// TIA Portal V17 export
// export: Created 2025-03-10T13:12:49.470688Z, ExportSetting WithDefaults, DisplayName Totally Integrated Automation Portal, DisplayVersion V17 Update 8, DisplayName TIA Portal Openness, DisplayVersion V17 Update 8, DisplayName TIA Portal Version Control Interface, DisplayVersion V17, DisplayName SINAMICS Startdrive Advanced, DisplayVersion V17 SP2, DisplayName SINAMICS Startdrive G110M, G120, G120C, G120D, G120P, G115D, DisplayVersion V17 SP2, DisplayName SINAMICS Startdrive G130, G150, S120, S150, SINAMICS MV, S210, DisplayVersion V17 SP2, DisplayName STEP 7 Professional, DisplayVersion V17 Update 8, DisplayName SINUMERIK ONE STEP 7 Toolbox, DisplayVersion V17 Update 12, DisplayName SINUMERIK 840D sl STEP 7 Toolbox, DisplayVersion V17 Update 12, DisplayName STEP 7 Safety, DisplayVersion V17 Update 6, DisplayName WinCC Advanced, DisplayVersion V17 Update 8
FUNCTION_BLOCK "FB21012_POWDER_FEEDER_HEATER_JKT"   // FB21012, LAD
TITLE = FB21012 POWDER FEEDER HEATER JKT
{ S7_Optimized_Access := 'FALSE' }
VERSION : 0.1
// stored: AutoNumber false, IsIECCheckEnabled false, SetENOAutomatically false, UDAEnableTagReadback false
   VAR_INPUT
      iPF_HEAT_AVAILABLE_OPTION : Bool;
      iPF_PROFINET_MODE_ACTIVE_FAULT : Bool;
      iPF_HOPPER_TEMP_GrHH_LINE_1 : Bool;   // POWDER FEEDER HOPPER TEMPERATURE LINE 1 ALARM
      iPF_HOPPER_TEMP_GrHH_LINE_2 : Bool;   // POWDER FEEDER HOPPER TEMPERATURE LINE 2 ALARM
      iCONTROL_ON_DELAYED : Bool;   // LOCAL MACHINE ON
      iAUTO_START_REQUEST : Bool;   // AUTO START REQUEST
      iAUTO_STOP_REQUEST : Bool;   // AUTO STOP SEQUEST
      iUNIT_NUMBER : Byte;
      iMANUAL_START_REQ_LINE_1 : Bool;
      iMANUAL_START_REQ_LINE_2 : Bool;
      iMANUAL_STOP_REQ_LINE_1 : Bool;
      iMANUAL_STOP_REQ_LINE_2 : Bool;
   END_VAR
   VAR_OUTPUT
      oPF_HEATING_ON_CMD_LINE_1 : Bool;   // POWDER FEEDER HEATING ON COMMAND LINE 1
      oPF_HEATING_ON_CMD_LINE_2 : Bool;   // POWDER FEEDER HEATING ON COMMAND LINE 2
      oPF_HEATING_OFF_CMD_LINE_1 : Bool;   // POWDER FEEDER HEATING OF COMMAND LINE 1
      oPF_HEATING_OFF_CMD_LINE_2 : Bool;   // POWDER FEEDER HEATING OF COMMAND LINE 2
      oSWITCHONCONDITION_ON_LINE_1 : Bool;
      oSWITCHONCONDITION_ON_LINE_2 : Bool;
      oSWITCHONCONDITION_OFF_LINE_1 : Bool;
      oSWITCHONCONDITION_OFF_LINE_2 : Bool;
      oMOTION_ACTIVE_RIGHT_LINE_1 : Bool;
      oMOTION_ACTIVE_RIGHT_LINE_2 : Bool;
      oMOTION_ACTIVE_LEFT_LINE_1 : Bool;
      oMOTION_ACTIVE_LEFT_LINE_2 : Bool;
      oLIMIT_RIGHT_LINE_1 : Bool;
      oLIMIT_RIGHT_LINE_2 : Bool;
      oLIMIT_LEFT_LINE_1 : Bool;
      oLIMIT_LEFT_LINE_2 : Bool;
      oALARM_HOPPER_LINE_1_TEMP_ABOVE_HIGH_LIMIT : Bool;
      oALARM_HOPPER_LINE_2_TEMP_ABOVE_HIGH_LIMIT : Bool;
   END_VAR
   VAR DB_SPECIFIC
      DATA : "POWDER FEEDER HEATER JKT";
      INPUT_SETTINGS : Struct
         UNIT_NUMBER : Int;
         FEEDER_NUMBER : Int;
      END_STRUCT;
      HEATER_STATUS_LINE_1 { S7_SetPoint := 'True'} : Byte;
      HEATER_STATUS_LINE_2 : Byte;
   END_VAR
   VAR_TEMP
      DB_NUMBER : DInt;
   END_VAR
   VAR_TEMP   // added for the SCL form of the ladder/FBD networks
      _w1 : Bool;
      _w2 : Bool;
   END_VAR
BEGIN

NETWORK
TITLE = READ INSTANCE DB NUMBER
      L     DINO;
      +     10#800000;
      T     #DB_NUMBER;

REGION Network 2: START GENERAL CONDITIONS / Start General Conditions
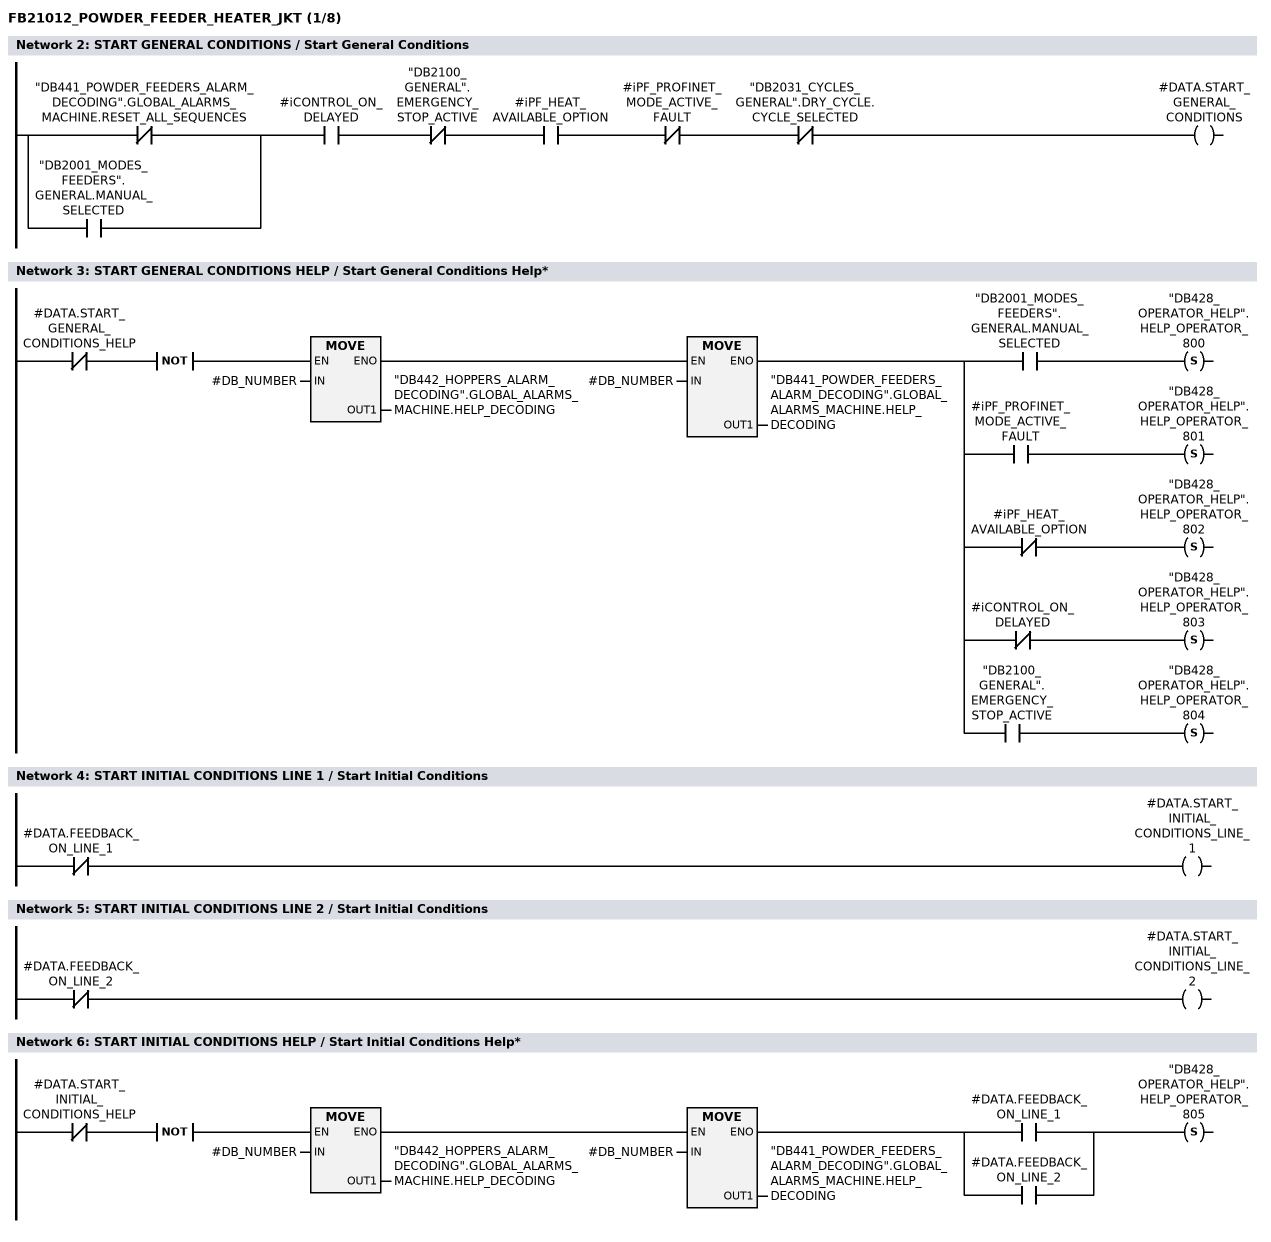
   RUNG wire#powerrail
      I_Contact( "DB441_POWDER_FEEDERS_ALARM_DECODING".GLOBAL_ALARMS_MACHINE.RESET_ALL_SEQUENCES )
      wire#w1
      Contact( #iCONTROL_ON_DELAYED )
      I_Contact( "DB2100_GENERAL".EMERGENCY_STOP_ACTIVE )
      Contact( #iPF_HEAT_AVAILABLE_OPTION )
      I_Contact( #iPF_PROFINET_MODE_ACTIVE_FAULT )
      I_Contact( "DB2031_CYCLES_GENERAL".DRY_CYCLE.CYCLE_SELECTED )
      Coil( #DATA.START_GENERAL_CONDITIONS )
   END_RUNG
   RUNG wire#powerrail
      Contact( "DB2001_MODES_FEEDERS".GENERAL.MANUAL_SELECTED )
   END_RUNG wire#w1
   // the same network as SCL:
   #DATA.START_GENERAL_CONDITIONS := (NOT "DB441_POWDER_FEEDERS_ALARM_DECODING".GLOBAL_ALARMS_MACHINE.RESET_ALL_SEQUENCES OR "DB2001_MODES_FEEDERS".GENERAL.MANUAL_SELECTED) AND #iCONTROL_ON_DELAYED AND NOT "DB2100_GENERAL".EMERGENCY_STOP_ACTIVE AND #iPF_HEAT_AVAILABLE_OPTION AND NOT #iPF_PROFINET_MODE_ACTIVE_FAULT AND NOT "DB2031_CYCLES_GENERAL".DRY_CYCLE.CYCLE_SELECTED;
END_REGION

REGION Network 3: START GENERAL CONDITIONS HELP / Start General Conditions Help*
   RUNG wire#powerrail
      I_Contact( #DATA.START_GENERAL_CONDITIONS_HELP )
      Not()
      Move(in := #DB_NUMBER, out1 => "DB442_HOPPERS_ALARM_DECODING".GLOBAL_ALARMS_MACHINE.HELP_DECODING)
      Move(in := #DB_NUMBER, out1 => "DB441_POWDER_FEEDERS_ALARM_DECODING".GLOBAL_ALARMS_MACHINE.HELP_DECODING)
      wire#w1
      Contact( "DB2001_MODES_FEEDERS".GENERAL.MANUAL_SELECTED )
      S_Coil( "DB428_OPERATOR_HELP".HELP_OPERATOR_800 )
   END_RUNG
   RUNG wire#w1
      Contact( #iPF_PROFINET_MODE_ACTIVE_FAULT )
      S_Coil( "DB428_OPERATOR_HELP".HELP_OPERATOR_801 )
   END_RUNG
   RUNG wire#w1
      I_Contact( #iPF_HEAT_AVAILABLE_OPTION )
      S_Coil( "DB428_OPERATOR_HELP".HELP_OPERATOR_802 )
   END_RUNG
   RUNG wire#w1
      I_Contact( #iCONTROL_ON_DELAYED )
      S_Coil( "DB428_OPERATOR_HELP".HELP_OPERATOR_803 )
   END_RUNG
   RUNG wire#w1
      Contact( "DB2100_GENERAL".EMERGENCY_STOP_ACTIVE )
      S_Coil( "DB428_OPERATOR_HELP".HELP_OPERATOR_804 )
   END_RUNG
   // the same network as SCL:
   #_w1 := NOT (NOT #DATA.START_GENERAL_CONDITIONS_HELP);
   IF #_w1 THEN
       "DB442_HOPPERS_ALARM_DECODING".GLOBAL_ALARMS_MACHINE.HELP_DECODING := #DB_NUMBER;
       "DB441_POWDER_FEEDERS_ALARM_DECODING".GLOBAL_ALARMS_MACHINE.HELP_DECODING := #DB_NUMBER;
   END_IF;
   IF #_w1 AND "DB2001_MODES_FEEDERS".GENERAL.MANUAL_SELECTED THEN
       "DB428_OPERATOR_HELP".HELP_OPERATOR_800 := TRUE;
   END_IF;
   IF #_w1 AND #iPF_PROFINET_MODE_ACTIVE_FAULT THEN "DB428_OPERATOR_HELP".HELP_OPERATOR_801 := TRUE; END_IF;
   IF #_w1 AND NOT #iPF_HEAT_AVAILABLE_OPTION THEN "DB428_OPERATOR_HELP".HELP_OPERATOR_802 := TRUE; END_IF;
   IF #_w1 AND NOT #iCONTROL_ON_DELAYED THEN "DB428_OPERATOR_HELP".HELP_OPERATOR_803 := TRUE; END_IF;
   IF #_w1 AND "DB2100_GENERAL".EMERGENCY_STOP_ACTIVE THEN
       "DB428_OPERATOR_HELP".HELP_OPERATOR_804 := TRUE;
   END_IF;
END_REGION

REGION Network 4: START INITIAL CONDITIONS LINE 1 / Start Initial Conditions
   RUNG wire#powerrail
      I_Contact( #DATA.FEEDBACK_ON_LINE_1 )
      Coil( #DATA.START_INITIAL_CONDITIONS_LINE_1 )
   END_RUNG
   // the same network as SCL:
   #DATA.START_INITIAL_CONDITIONS_LINE_1 := NOT #DATA.FEEDBACK_ON_LINE_1;
END_REGION

REGION Network 5: START INITIAL CONDITIONS LINE 2 / Start Initial Conditions
   RUNG wire#powerrail
      I_Contact( #DATA.FEEDBACK_ON_LINE_2 )
      Coil( #DATA.START_INITIAL_CONDITIONS_LINE_2 )
   END_RUNG
   // the same network as SCL:
   #DATA.START_INITIAL_CONDITIONS_LINE_2 := NOT #DATA.FEEDBACK_ON_LINE_2;
END_REGION

REGION Network 6: START INITIAL CONDITIONS HELP / Start Initial Conditions Help*
   RUNG wire#powerrail
      I_Contact( #DATA.START_INITIAL_CONDITIONS_HELP )
      Not()
      Move(in := #DB_NUMBER, out1 => "DB442_HOPPERS_ALARM_DECODING".GLOBAL_ALARMS_MACHINE.HELP_DECODING)
      Move(in := #DB_NUMBER, out1 => "DB441_POWDER_FEEDERS_ALARM_DECODING".GLOBAL_ALARMS_MACHINE.HELP_DECODING)
      wire#w1
      Contact( #DATA.FEEDBACK_ON_LINE_1 )
      wire#w2
      S_Coil( "DB428_OPERATOR_HELP".HELP_OPERATOR_805 )
   END_RUNG
   RUNG wire#w1
      Contact( #DATA.FEEDBACK_ON_LINE_2 )
   END_RUNG wire#w2
   // the same network as SCL:
   #_w1 := NOT (NOT #DATA.START_INITIAL_CONDITIONS_HELP);
   IF #_w1 THEN
       "DB442_HOPPERS_ALARM_DECODING".GLOBAL_ALARMS_MACHINE.HELP_DECODING := #DB_NUMBER;
       "DB441_POWDER_FEEDERS_ALARM_DECODING".GLOBAL_ALARMS_MACHINE.HELP_DECODING := #DB_NUMBER;
   END_IF;
   IF #_w1 AND (#DATA.FEEDBACK_ON_LINE_1 OR #DATA.FEEDBACK_ON_LINE_2) THEN
       "DB428_OPERATOR_HELP".HELP_OPERATOR_805 := TRUE;
   END_IF;
END_REGION

REGION Network 7: MANUAL MODE NOT SELECTED HELP / Manual Mode Not Selected Help*
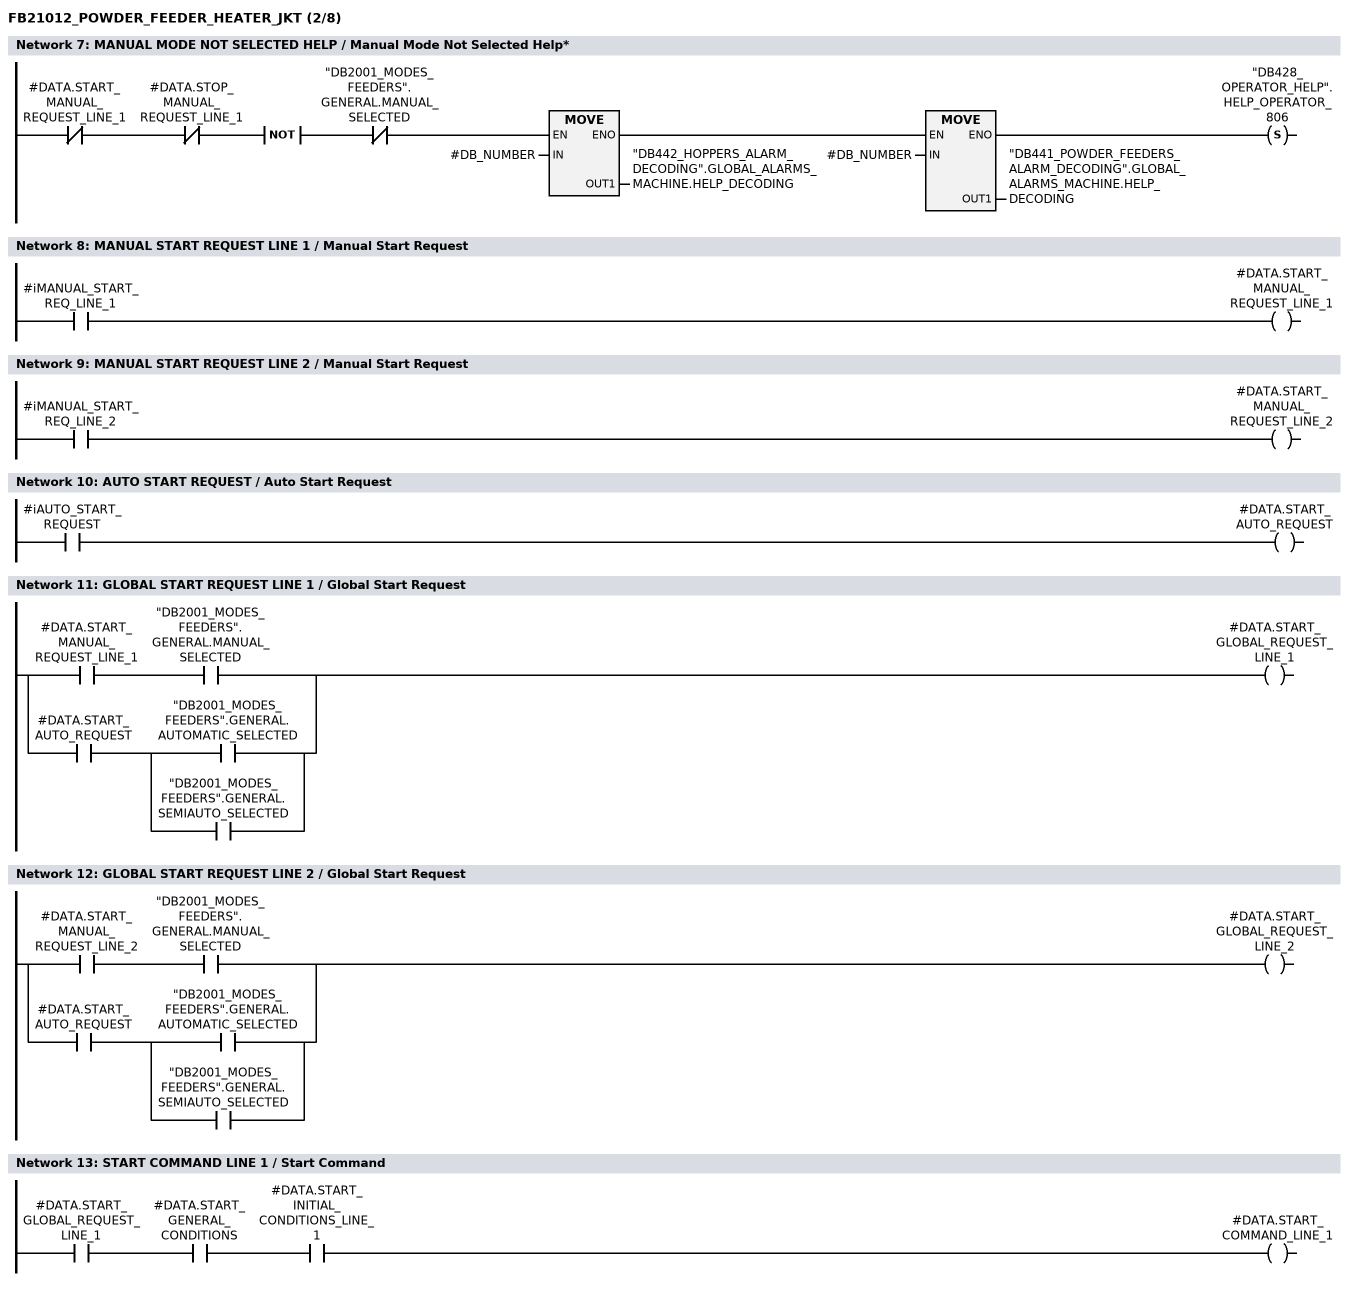
   RUNG wire#powerrail
      I_Contact( #DATA.START_MANUAL_REQUEST_LINE_1 )
      I_Contact( #DATA.STOP_MANUAL_REQUEST_LINE_1 )
      Not()
      I_Contact( "DB2001_MODES_FEEDERS".GENERAL.MANUAL_SELECTED )
      Move(in := #DB_NUMBER, out1 => "DB442_HOPPERS_ALARM_DECODING".GLOBAL_ALARMS_MACHINE.HELP_DECODING)
      Move(in := #DB_NUMBER, out1 => "DB441_POWDER_FEEDERS_ALARM_DECODING".GLOBAL_ALARMS_MACHINE.HELP_DECODING)
      S_Coil( "DB428_OPERATOR_HELP".HELP_OPERATOR_806 )
   END_RUNG
   // the same network as SCL:
   IF NOT (NOT #DATA.START_MANUAL_REQUEST_LINE_1 AND NOT #DATA.STOP_MANUAL_REQUEST_LINE_1) AND NOT "DB2001_MODES_FEEDERS".GENERAL.MANUAL_SELECTED THEN
       "DB442_HOPPERS_ALARM_DECODING".GLOBAL_ALARMS_MACHINE.HELP_DECODING := #DB_NUMBER;
       "DB441_POWDER_FEEDERS_ALARM_DECODING".GLOBAL_ALARMS_MACHINE.HELP_DECODING := #DB_NUMBER;
       "DB428_OPERATOR_HELP".HELP_OPERATOR_806 := TRUE;
   END_IF;
END_REGION

REGION Network 8: MANUAL START REQUEST LINE 1 / Manual Start Request
   RUNG wire#powerrail
      Contact( #iMANUAL_START_REQ_LINE_1 )
      Coil( #DATA.START_MANUAL_REQUEST_LINE_1 )
   END_RUNG
   // the same network as SCL:
   #DATA.START_MANUAL_REQUEST_LINE_1 := #iMANUAL_START_REQ_LINE_1;
END_REGION

REGION Network 9: MANUAL START REQUEST LINE 2 / Manual Start Request
   RUNG wire#powerrail
      Contact( #iMANUAL_START_REQ_LINE_2 )
      Coil( #DATA.START_MANUAL_REQUEST_LINE_2 )
   END_RUNG
   // the same network as SCL:
   #DATA.START_MANUAL_REQUEST_LINE_2 := #iMANUAL_START_REQ_LINE_2;
END_REGION

REGION Network 10: AUTO START REQUEST / Auto Start Request
   RUNG wire#powerrail
      Contact( #iAUTO_START_REQUEST )
      Coil( #DATA.START_AUTO_REQUEST )
   END_RUNG
   // the same network as SCL:
   #DATA.START_AUTO_REQUEST := #iAUTO_START_REQUEST;
END_REGION

REGION Network 11: GLOBAL START REQUEST LINE 1 / Global Start Request
   RUNG wire#powerrail
      Contact( #DATA.START_MANUAL_REQUEST_LINE_1 )
      Contact( "DB2001_MODES_FEEDERS".GENERAL.MANUAL_SELECTED )
      wire#w1
      Coil( #DATA.START_GLOBAL_REQUEST_LINE_1 )
   END_RUNG
   RUNG wire#powerrail
      Contact( #DATA.START_AUTO_REQUEST )
      wire#w2
      Contact( "DB2001_MODES_FEEDERS".GENERAL.AUTOMATIC_SELECTED )
   END_RUNG wire#w1
   RUNG wire#w2
      Contact( "DB2001_MODES_FEEDERS".GENERAL.SEMIAUTO_SELECTED )
   END_RUNG wire#w1
   // the same network as SCL:
   #DATA.START_GLOBAL_REQUEST_LINE_1 := (#DATA.START_MANUAL_REQUEST_LINE_1 AND "DB2001_MODES_FEEDERS".GENERAL.MANUAL_SELECTED) OR (#DATA.START_AUTO_REQUEST AND ("DB2001_MODES_FEEDERS".GENERAL.AUTOMATIC_SELECTED OR "DB2001_MODES_FEEDERS".GENERAL.SEMIAUTO_SELECTED));
END_REGION

REGION Network 12: GLOBAL START REQUEST LINE 2 / Global Start Request
   RUNG wire#powerrail
      Contact( #DATA.START_MANUAL_REQUEST_LINE_2 )
      Contact( "DB2001_MODES_FEEDERS".GENERAL.MANUAL_SELECTED )
      wire#w1
      Coil( #DATA.START_GLOBAL_REQUEST_LINE_2 )
   END_RUNG
   RUNG wire#powerrail
      Contact( #DATA.START_AUTO_REQUEST )
      wire#w2
      Contact( "DB2001_MODES_FEEDERS".GENERAL.AUTOMATIC_SELECTED )
   END_RUNG wire#w1
   RUNG wire#w2
      Contact( "DB2001_MODES_FEEDERS".GENERAL.SEMIAUTO_SELECTED )
   END_RUNG wire#w1
   // the same network as SCL:
   #DATA.START_GLOBAL_REQUEST_LINE_2 := (#DATA.START_MANUAL_REQUEST_LINE_2 AND "DB2001_MODES_FEEDERS".GENERAL.MANUAL_SELECTED) OR (#DATA.START_AUTO_REQUEST AND ("DB2001_MODES_FEEDERS".GENERAL.AUTOMATIC_SELECTED OR "DB2001_MODES_FEEDERS".GENERAL.SEMIAUTO_SELECTED));
END_REGION

REGION Network 13: START COMMAND LINE 1 / Start Command
   RUNG wire#powerrail
      Contact( #DATA.START_GLOBAL_REQUEST_LINE_1 )
      Contact( #DATA.START_GENERAL_CONDITIONS )
      Contact( #DATA.START_INITIAL_CONDITIONS_LINE_1 )
      Coil( #DATA.START_COMMAND_LINE_1 )
   END_RUNG
   // the same network as SCL:
   #DATA.START_COMMAND_LINE_1 := #DATA.START_GLOBAL_REQUEST_LINE_1 AND #DATA.START_GENERAL_CONDITIONS AND #DATA.START_INITIAL_CONDITIONS_LINE_1;
END_REGION

REGION Network 14: START COMMAND LINE 2 / Start Command
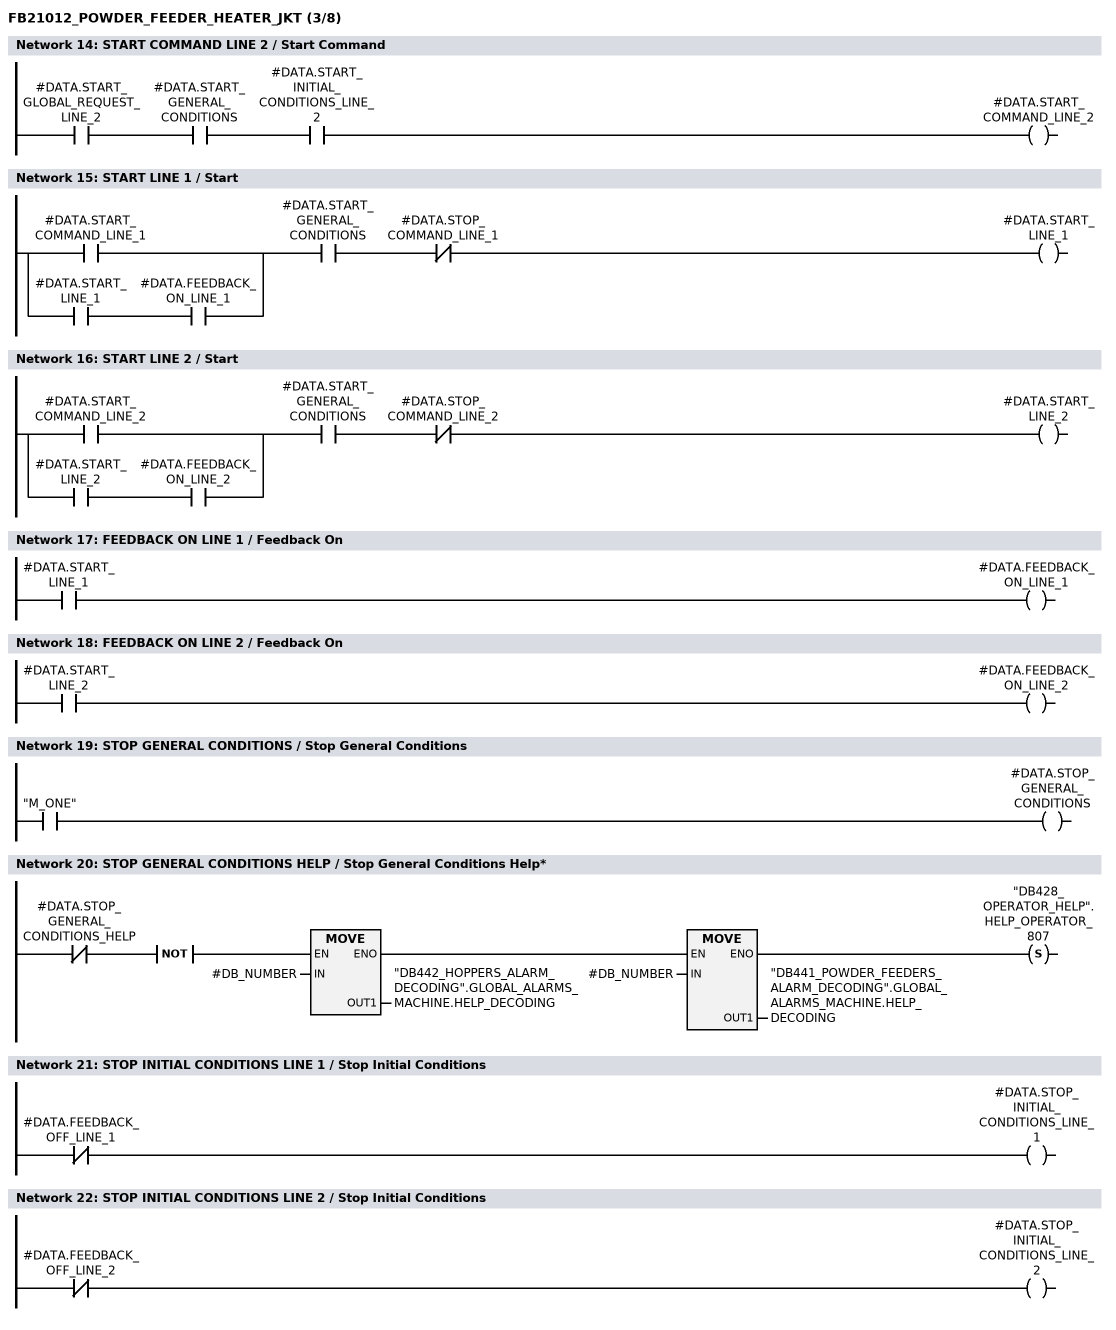
   RUNG wire#powerrail
      Contact( #DATA.START_GLOBAL_REQUEST_LINE_2 )
      Contact( #DATA.START_GENERAL_CONDITIONS )
      Contact( #DATA.START_INITIAL_CONDITIONS_LINE_2 )
      Coil( #DATA.START_COMMAND_LINE_2 )
   END_RUNG
   // the same network as SCL:
   #DATA.START_COMMAND_LINE_2 := #DATA.START_GLOBAL_REQUEST_LINE_2 AND #DATA.START_GENERAL_CONDITIONS AND #DATA.START_INITIAL_CONDITIONS_LINE_2;
END_REGION

REGION Network 15: START LINE 1 / Start
   RUNG wire#powerrail
      Contact( #DATA.START_COMMAND_LINE_1 )
      wire#w1
      Contact( #DATA.START_GENERAL_CONDITIONS )
      I_Contact( #DATA.STOP_COMMAND_LINE_1 )
      Coil( #DATA.START_LINE_1 )
   END_RUNG
   RUNG wire#powerrail
      Contact( #DATA.START_LINE_1 )
      Contact( #DATA.FEEDBACK_ON_LINE_1 )
   END_RUNG wire#w1
   // the same network as SCL:
   #DATA.START_LINE_1 := (#DATA.START_COMMAND_LINE_1 OR (#DATA.START_LINE_1 AND #DATA.FEEDBACK_ON_LINE_1)) AND #DATA.START_GENERAL_CONDITIONS AND NOT #DATA.STOP_COMMAND_LINE_1;
END_REGION

REGION Network 16: START LINE 2 / Start
   RUNG wire#powerrail
      Contact( #DATA.START_COMMAND_LINE_2 )
      wire#w1
      Contact( #DATA.START_GENERAL_CONDITIONS )
      I_Contact( #DATA.STOP_COMMAND_LINE_2 )
      Coil( #DATA.START_LINE_2 )
   END_RUNG
   RUNG wire#powerrail
      Contact( #DATA.START_LINE_2 )
      Contact( #DATA.FEEDBACK_ON_LINE_2 )
   END_RUNG wire#w1
   // the same network as SCL:
   #DATA.START_LINE_2 := (#DATA.START_COMMAND_LINE_2 OR (#DATA.START_LINE_2 AND #DATA.FEEDBACK_ON_LINE_2)) AND #DATA.START_GENERAL_CONDITIONS AND NOT #DATA.STOP_COMMAND_LINE_2;
END_REGION

REGION Network 17: FEEDBACK ON LINE 1 / Feedback On
   RUNG wire#powerrail
      Contact( #DATA.START_LINE_1 )
      Coil( #DATA.FEEDBACK_ON_LINE_1 )
   END_RUNG
   // the same network as SCL:
   #DATA.FEEDBACK_ON_LINE_1 := #DATA.START_LINE_1;
END_REGION

REGION Network 18: FEEDBACK ON LINE 2 / Feedback On
   RUNG wire#powerrail
      Contact( #DATA.START_LINE_2 )
      Coil( #DATA.FEEDBACK_ON_LINE_2 )
   END_RUNG
   // the same network as SCL:
   #DATA.FEEDBACK_ON_LINE_2 := #DATA.START_LINE_2;
END_REGION

REGION Network 19: STOP GENERAL CONDITIONS / Stop General Conditions
   RUNG wire#powerrail
      Contact( "M_ONE" )
      Coil( #DATA.STOP_GENERAL_CONDITIONS )
   END_RUNG
   // the same network as SCL:
   #DATA.STOP_GENERAL_CONDITIONS := "M_ONE";
END_REGION

REGION Network 20: STOP GENERAL CONDITIONS HELP / Stop General Conditions Help*
   RUNG wire#powerrail
      I_Contact( #DATA.STOP_GENERAL_CONDITIONS_HELP )
      Not()
      Move(in := #DB_NUMBER, out1 => "DB442_HOPPERS_ALARM_DECODING".GLOBAL_ALARMS_MACHINE.HELP_DECODING)
      Move(in := #DB_NUMBER, out1 => "DB441_POWDER_FEEDERS_ALARM_DECODING".GLOBAL_ALARMS_MACHINE.HELP_DECODING)
      S_Coil( "DB428_OPERATOR_HELP".HELP_OPERATOR_807 )
   END_RUNG
   // the same network as SCL:
   IF NOT (NOT #DATA.STOP_GENERAL_CONDITIONS_HELP) THEN
       "DB442_HOPPERS_ALARM_DECODING".GLOBAL_ALARMS_MACHINE.HELP_DECODING := #DB_NUMBER;
       "DB441_POWDER_FEEDERS_ALARM_DECODING".GLOBAL_ALARMS_MACHINE.HELP_DECODING := #DB_NUMBER;
       "DB428_OPERATOR_HELP".HELP_OPERATOR_807 := TRUE;
   END_IF;
END_REGION

REGION Network 21: STOP INITIAL CONDITIONS LINE 1 / Stop Initial Conditions
   RUNG wire#powerrail
      I_Contact( #DATA.FEEDBACK_OFF_LINE_1 )
      Coil( #DATA.STOP_INITIAL_CONDITIONS_LINE_1 )
   END_RUNG
   // the same network as SCL:
   #DATA.STOP_INITIAL_CONDITIONS_LINE_1 := NOT #DATA.FEEDBACK_OFF_LINE_1;
END_REGION

REGION Network 22: STOP INITIAL CONDITIONS LINE 2 / Stop Initial Conditions
   RUNG wire#powerrail
      I_Contact( #DATA.FEEDBACK_OFF_LINE_2 )
      Coil( #DATA.STOP_INITIAL_CONDITIONS_LINE_2 )
   END_RUNG
   // the same network as SCL:
   #DATA.STOP_INITIAL_CONDITIONS_LINE_2 := NOT #DATA.FEEDBACK_OFF_LINE_2;
END_REGION

REGION Network 23: STOP INITIAL CONDITIONS HELP / Stop Initial Conditions Help*
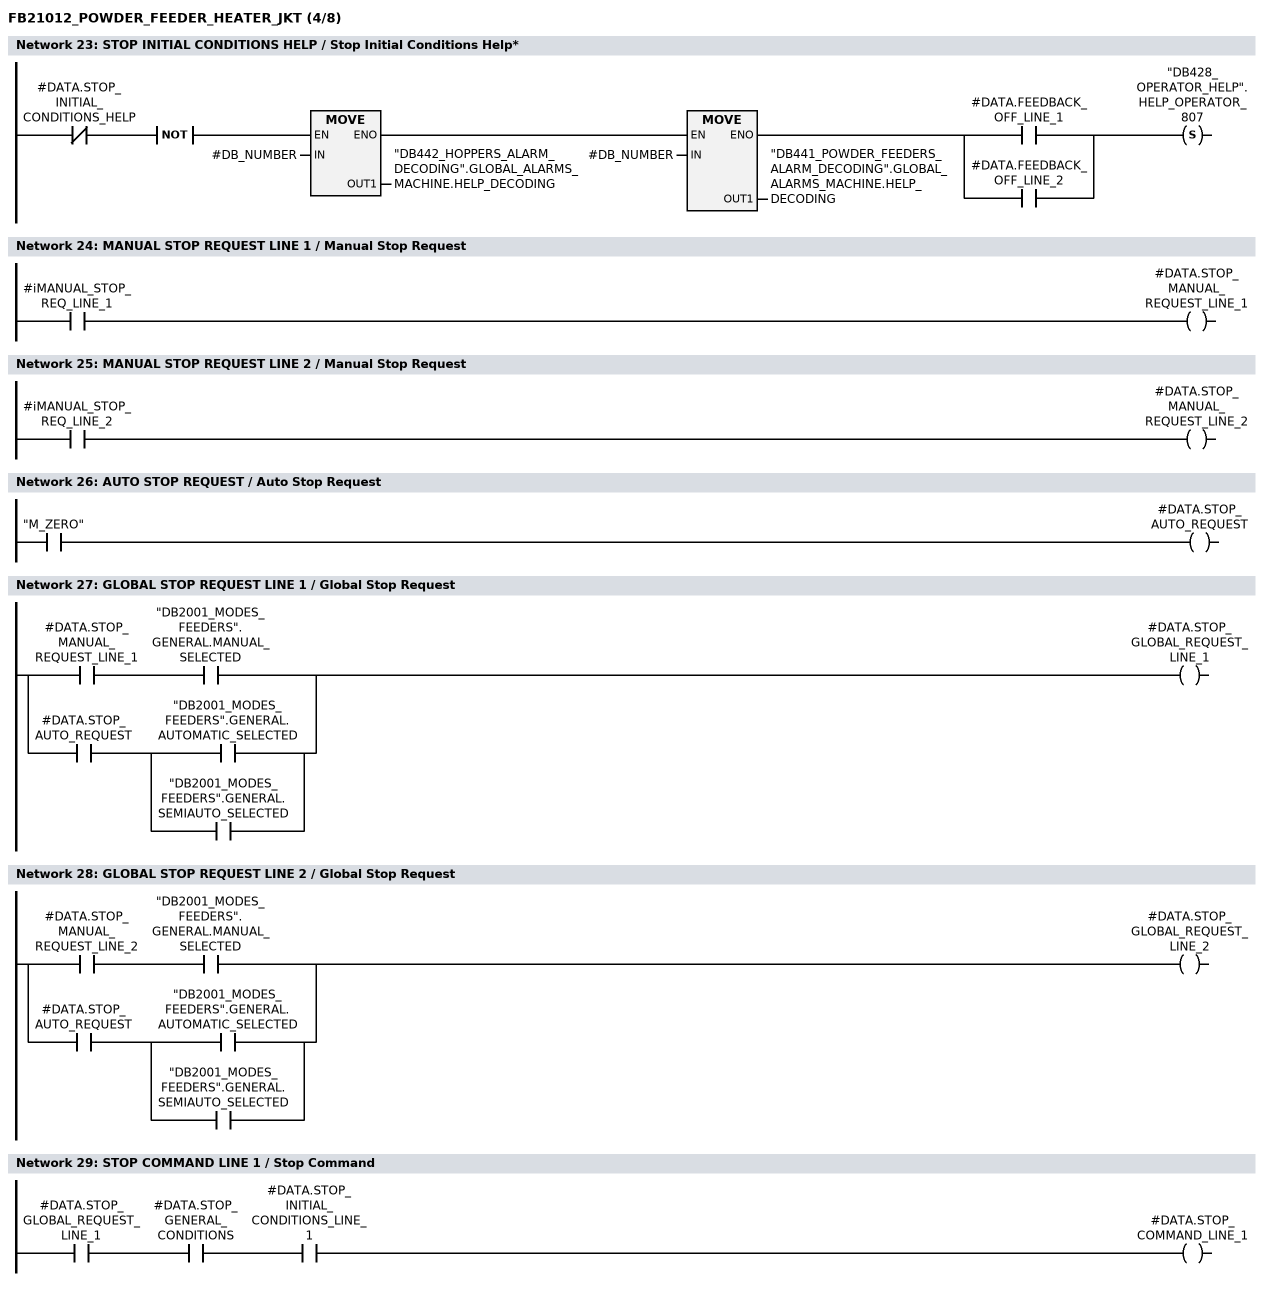
   RUNG wire#powerrail
      I_Contact( #DATA.STOP_INITIAL_CONDITIONS_HELP )
      Not()
      Move(in := #DB_NUMBER, out1 => "DB442_HOPPERS_ALARM_DECODING".GLOBAL_ALARMS_MACHINE.HELP_DECODING)
      Move(in := #DB_NUMBER, out1 => "DB441_POWDER_FEEDERS_ALARM_DECODING".GLOBAL_ALARMS_MACHINE.HELP_DECODING)
      wire#w1
      Contact( #DATA.FEEDBACK_OFF_LINE_1 )
      wire#w2
      S_Coil( "DB428_OPERATOR_HELP".HELP_OPERATOR_807 )
   END_RUNG
   RUNG wire#w1
      Contact( #DATA.FEEDBACK_OFF_LINE_2 )
   END_RUNG wire#w2
   // the same network as SCL:
   #_w1 := NOT (NOT #DATA.STOP_INITIAL_CONDITIONS_HELP);
   IF #_w1 THEN
       "DB442_HOPPERS_ALARM_DECODING".GLOBAL_ALARMS_MACHINE.HELP_DECODING := #DB_NUMBER;
       "DB441_POWDER_FEEDERS_ALARM_DECODING".GLOBAL_ALARMS_MACHINE.HELP_DECODING := #DB_NUMBER;
   END_IF;
   IF #_w1 AND (#DATA.FEEDBACK_OFF_LINE_1 OR #DATA.FEEDBACK_OFF_LINE_2) THEN
       "DB428_OPERATOR_HELP".HELP_OPERATOR_807 := TRUE;
   END_IF;
END_REGION

REGION Network 24: MANUAL STOP REQUEST LINE 1 / Manual Stop Request
   RUNG wire#powerrail
      Contact( #iMANUAL_STOP_REQ_LINE_1 )
      Coil( #DATA.STOP_MANUAL_REQUEST_LINE_1 )
   END_RUNG
   // the same network as SCL:
   #DATA.STOP_MANUAL_REQUEST_LINE_1 := #iMANUAL_STOP_REQ_LINE_1;
END_REGION

REGION Network 25: MANUAL STOP REQUEST LINE 2 / Manual Stop Request
   RUNG wire#powerrail
      Contact( #iMANUAL_STOP_REQ_LINE_2 )
      Coil( #DATA.STOP_MANUAL_REQUEST_LINE_2 )
   END_RUNG
   // the same network as SCL:
   #DATA.STOP_MANUAL_REQUEST_LINE_2 := #iMANUAL_STOP_REQ_LINE_2;
END_REGION

REGION Network 26: AUTO STOP REQUEST / Auto Stop Request
   RUNG wire#powerrail
      Contact( "M_ZERO" )
      Coil( #DATA.STOP_AUTO_REQUEST )
   END_RUNG
   // the same network as SCL:
   #DATA.STOP_AUTO_REQUEST := "M_ZERO";
END_REGION

REGION Network 27: GLOBAL STOP REQUEST LINE 1 / Global Stop Request
   RUNG wire#powerrail
      Contact( #DATA.STOP_MANUAL_REQUEST_LINE_1 )
      Contact( "DB2001_MODES_FEEDERS".GENERAL.MANUAL_SELECTED )
      wire#w1
      Coil( #DATA.STOP_GLOBAL_REQUEST_LINE_1 )
   END_RUNG
   RUNG wire#powerrail
      Contact( #DATA.STOP_AUTO_REQUEST )
      wire#w2
      Contact( "DB2001_MODES_FEEDERS".GENERAL.AUTOMATIC_SELECTED )
   END_RUNG wire#w1
   RUNG wire#w2
      Contact( "DB2001_MODES_FEEDERS".GENERAL.SEMIAUTO_SELECTED )
   END_RUNG wire#w1
   // the same network as SCL:
   #DATA.STOP_GLOBAL_REQUEST_LINE_1 := (#DATA.STOP_MANUAL_REQUEST_LINE_1 AND "DB2001_MODES_FEEDERS".GENERAL.MANUAL_SELECTED) OR (#DATA.STOP_AUTO_REQUEST AND ("DB2001_MODES_FEEDERS".GENERAL.AUTOMATIC_SELECTED OR "DB2001_MODES_FEEDERS".GENERAL.SEMIAUTO_SELECTED));
END_REGION

REGION Network 28: GLOBAL STOP REQUEST LINE 2 / Global Stop Request
   RUNG wire#powerrail
      Contact( #DATA.STOP_MANUAL_REQUEST_LINE_2 )
      Contact( "DB2001_MODES_FEEDERS".GENERAL.MANUAL_SELECTED )
      wire#w1
      Coil( #DATA.STOP_GLOBAL_REQUEST_LINE_2 )
   END_RUNG
   RUNG wire#powerrail
      Contact( #DATA.STOP_AUTO_REQUEST )
      wire#w2
      Contact( "DB2001_MODES_FEEDERS".GENERAL.AUTOMATIC_SELECTED )
   END_RUNG wire#w1
   RUNG wire#w2
      Contact( "DB2001_MODES_FEEDERS".GENERAL.SEMIAUTO_SELECTED )
   END_RUNG wire#w1
   // the same network as SCL:
   #DATA.STOP_GLOBAL_REQUEST_LINE_2 := (#DATA.STOP_MANUAL_REQUEST_LINE_2 AND "DB2001_MODES_FEEDERS".GENERAL.MANUAL_SELECTED) OR (#DATA.STOP_AUTO_REQUEST AND ("DB2001_MODES_FEEDERS".GENERAL.AUTOMATIC_SELECTED OR "DB2001_MODES_FEEDERS".GENERAL.SEMIAUTO_SELECTED));
END_REGION

REGION Network 29: STOP COMMAND LINE 1 / Stop Command
   RUNG wire#powerrail
      Contact( #DATA.STOP_GLOBAL_REQUEST_LINE_1 )
      Contact( #DATA.STOP_GENERAL_CONDITIONS )
      Contact( #DATA.STOP_INITIAL_CONDITIONS_LINE_1 )
      Coil( #DATA.STOP_COMMAND_LINE_1 )
   END_RUNG
   // the same network as SCL:
   #DATA.STOP_COMMAND_LINE_1 := #DATA.STOP_GLOBAL_REQUEST_LINE_1 AND #DATA.STOP_GENERAL_CONDITIONS AND #DATA.STOP_INITIAL_CONDITIONS_LINE_1;
END_REGION

REGION Network 30: STOP COMMAND LINE 2 / Stop Command
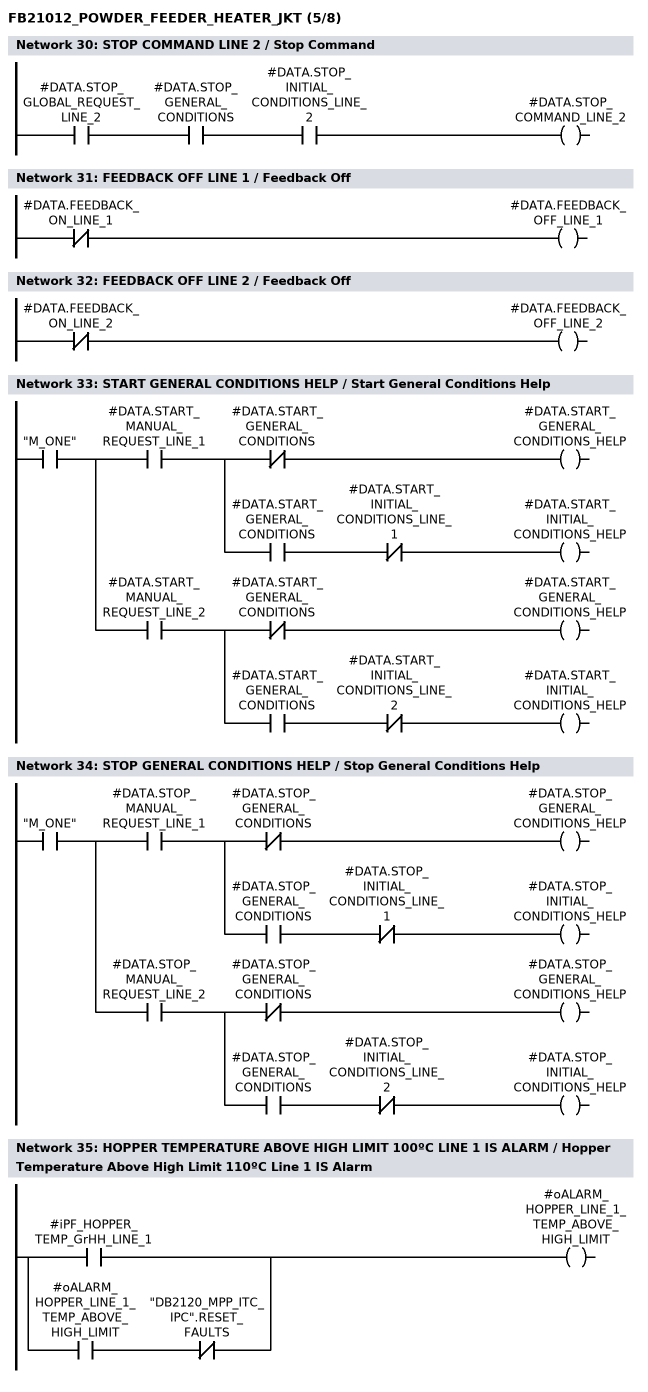
   RUNG wire#powerrail
      Contact( #DATA.STOP_GLOBAL_REQUEST_LINE_2 )
      Contact( #DATA.STOP_GENERAL_CONDITIONS )
      Contact( #DATA.STOP_INITIAL_CONDITIONS_LINE_2 )
      Coil( #DATA.STOP_COMMAND_LINE_2 )
   END_RUNG
   // the same network as SCL:
   #DATA.STOP_COMMAND_LINE_2 := #DATA.STOP_GLOBAL_REQUEST_LINE_2 AND #DATA.STOP_GENERAL_CONDITIONS AND #DATA.STOP_INITIAL_CONDITIONS_LINE_2;
END_REGION

REGION Network 31: FEEDBACK OFF LINE 1 / Feedback Off
   RUNG wire#powerrail
      I_Contact( #DATA.FEEDBACK_ON_LINE_1 )
      Coil( #DATA.FEEDBACK_OFF_LINE_1 )
   END_RUNG
   // the same network as SCL:
   #DATA.FEEDBACK_OFF_LINE_1 := NOT #DATA.FEEDBACK_ON_LINE_1;
END_REGION

REGION Network 32: FEEDBACK OFF LINE 2 / Feedback Off
   RUNG wire#powerrail
      I_Contact( #DATA.FEEDBACK_ON_LINE_2 )
      Coil( #DATA.FEEDBACK_OFF_LINE_2 )
   END_RUNG
   // the same network as SCL:
   #DATA.FEEDBACK_OFF_LINE_2 := NOT #DATA.FEEDBACK_ON_LINE_2;
END_REGION

REGION Network 33: START GENERAL CONDITIONS HELP / Start General Conditions Help
   RUNG wire#powerrail
      Contact( "M_ONE" )
      wire#w1
      Contact( #DATA.START_MANUAL_REQUEST_LINE_1 )
      wire#w2
      I_Contact( #DATA.START_GENERAL_CONDITIONS )
      Coil( #DATA.START_GENERAL_CONDITIONS_HELP )
   END_RUNG
   RUNG wire#w2
      Contact( #DATA.START_GENERAL_CONDITIONS )
      I_Contact( #DATA.START_INITIAL_CONDITIONS_LINE_1 )
      Coil( #DATA.START_INITIAL_CONDITIONS_HELP )
   END_RUNG
   RUNG wire#w1
      Contact( #DATA.START_MANUAL_REQUEST_LINE_2 )
      wire#w3
      I_Contact( #DATA.START_GENERAL_CONDITIONS )
      Coil( #DATA.START_GENERAL_CONDITIONS_HELP )
   END_RUNG
   RUNG wire#w3
      Contact( #DATA.START_GENERAL_CONDITIONS )
      I_Contact( #DATA.START_INITIAL_CONDITIONS_LINE_2 )
      Coil( #DATA.START_INITIAL_CONDITIONS_HELP )
   END_RUNG
   // the same network as SCL:
   #_w1 := "M_ONE" AND #DATA.START_MANUAL_REQUEST_LINE_1;
   #DATA.START_GENERAL_CONDITIONS_HELP := #_w1 AND NOT #DATA.START_GENERAL_CONDITIONS;
   #DATA.START_INITIAL_CONDITIONS_HELP := #_w1 AND #DATA.START_GENERAL_CONDITIONS AND NOT #DATA.START_INITIAL_CONDITIONS_LINE_1;
   #_w2 := "M_ONE" AND #DATA.START_MANUAL_REQUEST_LINE_2;
   #DATA.START_GENERAL_CONDITIONS_HELP := #_w2 AND NOT #DATA.START_GENERAL_CONDITIONS;
   #DATA.START_INITIAL_CONDITIONS_HELP := #_w2 AND #DATA.START_GENERAL_CONDITIONS AND NOT #DATA.START_INITIAL_CONDITIONS_LINE_2;
END_REGION

REGION Network 34: STOP GENERAL CONDITIONS HELP / Stop General Conditions Help
   RUNG wire#powerrail
      Contact( "M_ONE" )
      wire#w1
      Contact( #DATA.STOP_MANUAL_REQUEST_LINE_1 )
      wire#w2
      I_Contact( #DATA.STOP_GENERAL_CONDITIONS )
      Coil( #DATA.STOP_GENERAL_CONDITIONS_HELP )
   END_RUNG
   RUNG wire#w2
      Contact( #DATA.STOP_GENERAL_CONDITIONS )
      I_Contact( #DATA.STOP_INITIAL_CONDITIONS_LINE_1 )
      Coil( #DATA.STOP_INITIAL_CONDITIONS_HELP )
   END_RUNG
   RUNG wire#w1
      Contact( #DATA.STOP_MANUAL_REQUEST_LINE_2 )
      wire#w3
      I_Contact( #DATA.STOP_GENERAL_CONDITIONS )
      Coil( #DATA.STOP_GENERAL_CONDITIONS_HELP )
   END_RUNG
   RUNG wire#w3
      Contact( #DATA.STOP_GENERAL_CONDITIONS )
      I_Contact( #DATA.STOP_INITIAL_CONDITIONS_LINE_2 )
      Coil( #DATA.STOP_INITIAL_CONDITIONS_HELP )
   END_RUNG
   // the same network as SCL:
   #_w1 := "M_ONE" AND #DATA.STOP_MANUAL_REQUEST_LINE_1;
   #DATA.STOP_GENERAL_CONDITIONS_HELP := #_w1 AND NOT #DATA.STOP_GENERAL_CONDITIONS;
   #DATA.STOP_INITIAL_CONDITIONS_HELP := #_w1 AND #DATA.STOP_GENERAL_CONDITIONS AND NOT #DATA.STOP_INITIAL_CONDITIONS_LINE_1;
   #_w2 := "M_ONE" AND #DATA.STOP_MANUAL_REQUEST_LINE_2;
   #DATA.STOP_GENERAL_CONDITIONS_HELP := #_w2 AND NOT #DATA.STOP_GENERAL_CONDITIONS;
   #DATA.STOP_INITIAL_CONDITIONS_HELP := #_w2 AND #DATA.STOP_GENERAL_CONDITIONS AND NOT #DATA.STOP_INITIAL_CONDITIONS_LINE_2;
END_REGION

REGION Network 35: HOPPER TEMPERATURE ABOVE HIGH LIMIT 100ºC LINE 1 IS ALARM / Hopper Temperature Above High Limit 110ºC Line 1 IS Alarm
   RUNG wire#powerrail
      Contact( #iPF_HOPPER_TEMP_GrHH_LINE_1 )
      wire#w1
      Coil( #oALARM_HOPPER_LINE_1_TEMP_ABOVE_HIGH_LIMIT )
   END_RUNG
   RUNG wire#powerrail
      Contact( #oALARM_HOPPER_LINE_1_TEMP_ABOVE_HIGH_LIMIT )
      I_Contact( "DB2120_MPP_ITC_IPC".RESET_FAULTS )
   END_RUNG wire#w1
   // the same network as SCL:
   #oALARM_HOPPER_LINE_1_TEMP_ABOVE_HIGH_LIMIT := #iPF_HOPPER_TEMP_GrHH_LINE_1 OR (#oALARM_HOPPER_LINE_1_TEMP_ABOVE_HIGH_LIMIT AND NOT "DB2120_MPP_ITC_IPC".RESET_FAULTS);
END_REGION

REGION Network 36: HOPPER TEMPERATURE ABOVE HIGH LIMIT 100ºC LINE 2 IS ALARM / Hopper Temperature Above High Limit 110ºC Line 1 IS Alarm
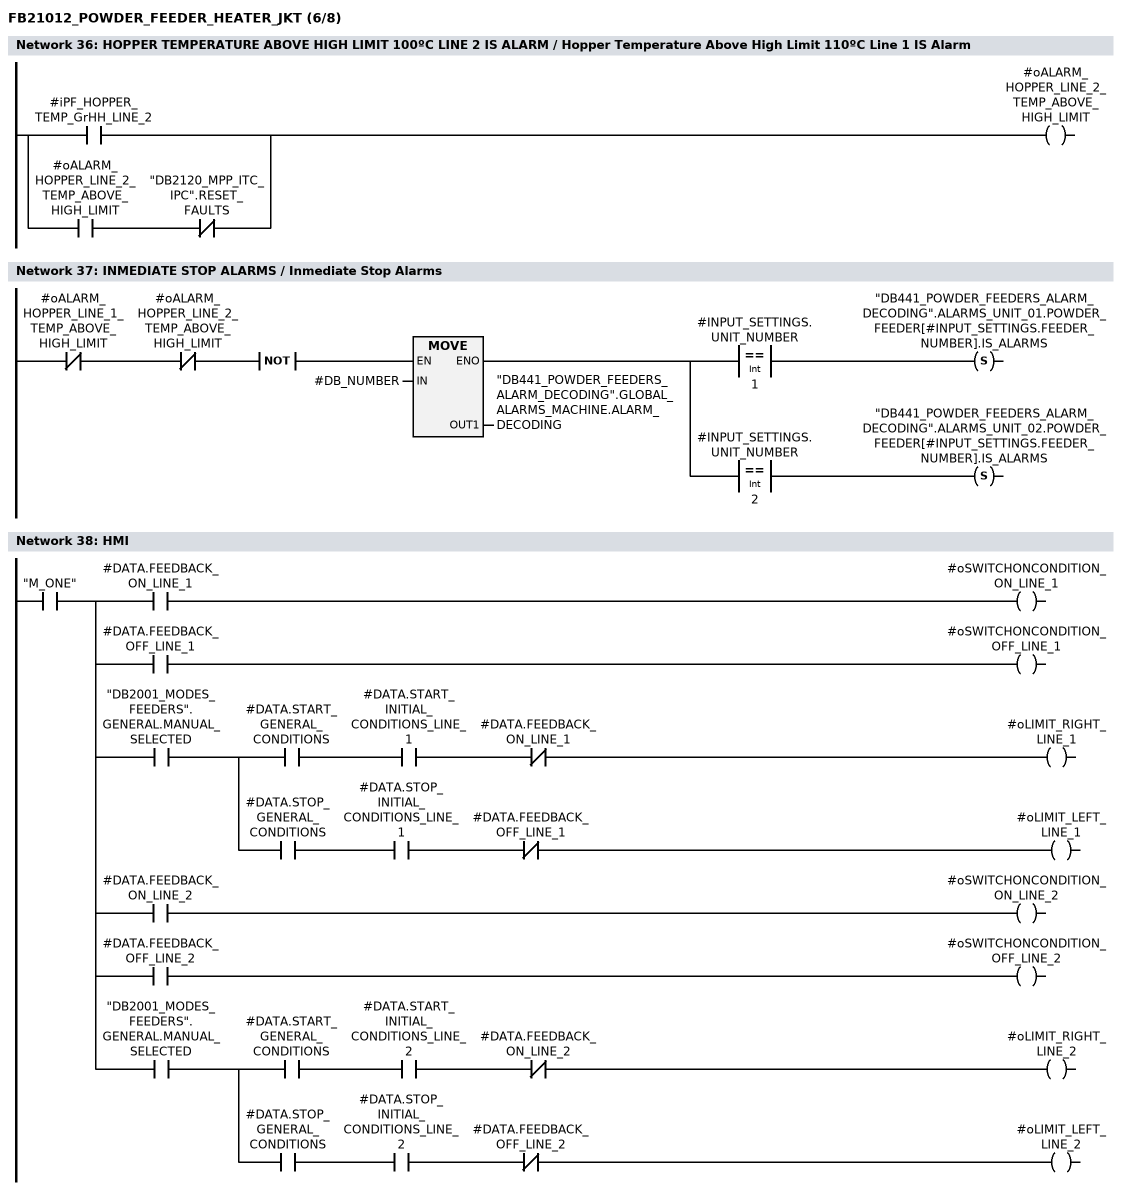
   RUNG wire#powerrail
      Contact( #iPF_HOPPER_TEMP_GrHH_LINE_2 )
      wire#w1
      Coil( #oALARM_HOPPER_LINE_2_TEMP_ABOVE_HIGH_LIMIT )
   END_RUNG
   RUNG wire#powerrail
      Contact( #oALARM_HOPPER_LINE_2_TEMP_ABOVE_HIGH_LIMIT )
      I_Contact( "DB2120_MPP_ITC_IPC".RESET_FAULTS )
   END_RUNG wire#w1
   // the same network as SCL:
   #oALARM_HOPPER_LINE_2_TEMP_ABOVE_HIGH_LIMIT := #iPF_HOPPER_TEMP_GrHH_LINE_2 OR (#oALARM_HOPPER_LINE_2_TEMP_ABOVE_HIGH_LIMIT AND NOT "DB2120_MPP_ITC_IPC".RESET_FAULTS);
END_REGION

REGION Network 37: INMEDIATE STOP ALARMS / Inmediate Stop Alarms
   RUNG wire#powerrail
      I_Contact( #oALARM_HOPPER_LINE_1_TEMP_ABOVE_HIGH_LIMIT )
      I_Contact( #oALARM_HOPPER_LINE_2_TEMP_ABOVE_HIGH_LIMIT )
      Not()
      Move(in := #DB_NUMBER, out1 => "DB441_POWDER_FEEDERS_ALARM_DECODING".GLOBAL_ALARMS_MACHINE.ALARM_DECODING)
      wire#w1
      { S7_Templates := "SrcType := Int" } EQ_Contact(in1 := #INPUT_SETTINGS.UNIT_NUMBER, in2 := 1)
      S_Coil( "DB441_POWDER_FEEDERS_ALARM_DECODING".ALARMS_UNIT_01.POWDER_FEEDER[#INPUT_SETTINGS.FEEDER_NUMBER].IS_ALARMS )
   END_RUNG
   RUNG wire#w1
      { S7_Templates := "SrcType := Int" } EQ_Contact(in1 := #INPUT_SETTINGS.UNIT_NUMBER, in2 := 2)
      S_Coil( "DB441_POWDER_FEEDERS_ALARM_DECODING".ALARMS_UNIT_02.POWDER_FEEDER[#INPUT_SETTINGS.FEEDER_NUMBER].IS_ALARMS )
   END_RUNG
   // the same network as SCL:
   #_w1 := NOT (NOT #oALARM_HOPPER_LINE_1_TEMP_ABOVE_HIGH_LIMIT AND NOT #oALARM_HOPPER_LINE_2_TEMP_ABOVE_HIGH_LIMIT);
   IF #_w1 THEN
       "DB441_POWDER_FEEDERS_ALARM_DECODING".GLOBAL_ALARMS_MACHINE.ALARM_DECODING := #DB_NUMBER;
   END_IF;
   IF #_w1 AND (#INPUT_SETTINGS.UNIT_NUMBER = 1) THEN
       "DB441_POWDER_FEEDERS_ALARM_DECODING".ALARMS_UNIT_01.POWDER_FEEDER[#INPUT_SETTINGS.FEEDER_NUMBER].IS_ALARMS := TRUE;
   END_IF;
   IF #_w1 AND (#INPUT_SETTINGS.UNIT_NUMBER = 2) THEN
       "DB441_POWDER_FEEDERS_ALARM_DECODING".ALARMS_UNIT_02.POWDER_FEEDER[#INPUT_SETTINGS.FEEDER_NUMBER].IS_ALARMS := TRUE;
   END_IF;
END_REGION

REGION Network 38: HMI
   RUNG wire#powerrail
      Contact( "M_ONE" )
      wire#w1
      Contact( #DATA.FEEDBACK_ON_LINE_1 )
      Coil( #oSWITCHONCONDITION_ON_LINE_1 )
   END_RUNG
   RUNG wire#w1
      Contact( #DATA.FEEDBACK_OFF_LINE_1 )
      Coil( #oSWITCHONCONDITION_OFF_LINE_1 )
   END_RUNG
   RUNG wire#w1
      Contact( "DB2001_MODES_FEEDERS".GENERAL.MANUAL_SELECTED )
      wire#w2
      Contact( #DATA.START_GENERAL_CONDITIONS )
      Contact( #DATA.START_INITIAL_CONDITIONS_LINE_1 )
      I_Contact( #DATA.FEEDBACK_ON_LINE_1 )
      Coil( #oLIMIT_RIGHT_LINE_1 )
   END_RUNG
   RUNG wire#w2
      Contact( #DATA.STOP_GENERAL_CONDITIONS )
      Contact( #DATA.STOP_INITIAL_CONDITIONS_LINE_1 )
      I_Contact( #DATA.FEEDBACK_OFF_LINE_1 )
      Coil( #oLIMIT_LEFT_LINE_1 )
   END_RUNG
   RUNG wire#w1
      Contact( #DATA.FEEDBACK_ON_LINE_2 )
      Coil( #oSWITCHONCONDITION_ON_LINE_2 )
   END_RUNG
   RUNG wire#w1
      Contact( #DATA.FEEDBACK_OFF_LINE_2 )
      Coil( #oSWITCHONCONDITION_OFF_LINE_2 )
   END_RUNG
   RUNG wire#w1
      Contact( "DB2001_MODES_FEEDERS".GENERAL.MANUAL_SELECTED )
      wire#w3
      Contact( #DATA.START_GENERAL_CONDITIONS )
      Contact( #DATA.START_INITIAL_CONDITIONS_LINE_2 )
      I_Contact( #DATA.FEEDBACK_ON_LINE_2 )
      Coil( #oLIMIT_RIGHT_LINE_2 )
   END_RUNG
   RUNG wire#w3
      Contact( #DATA.STOP_GENERAL_CONDITIONS )
      Contact( #DATA.STOP_INITIAL_CONDITIONS_LINE_2 )
      I_Contact( #DATA.FEEDBACK_OFF_LINE_2 )
      Coil( #oLIMIT_LEFT_LINE_2 )
   END_RUNG
   // the same network as SCL:
   #oSWITCHONCONDITION_ON_LINE_1 := "M_ONE" AND #DATA.FEEDBACK_ON_LINE_1;
   #oSWITCHONCONDITION_OFF_LINE_1 := "M_ONE" AND #DATA.FEEDBACK_OFF_LINE_1;
   #_w1 := "M_ONE" AND "DB2001_MODES_FEEDERS".GENERAL.MANUAL_SELECTED;
   #oLIMIT_RIGHT_LINE_1 := #_w1 AND #DATA.START_GENERAL_CONDITIONS AND #DATA.START_INITIAL_CONDITIONS_LINE_1 AND NOT #DATA.FEEDBACK_ON_LINE_1;
   #oLIMIT_LEFT_LINE_1 := #_w1 AND #DATA.STOP_GENERAL_CONDITIONS AND #DATA.STOP_INITIAL_CONDITIONS_LINE_1 AND NOT #DATA.FEEDBACK_OFF_LINE_1;
   #oSWITCHONCONDITION_ON_LINE_2 := "M_ONE" AND #DATA.FEEDBACK_ON_LINE_2;
   #oSWITCHONCONDITION_OFF_LINE_2 := "M_ONE" AND #DATA.FEEDBACK_OFF_LINE_2;
   #_w2 := "M_ONE" AND "DB2001_MODES_FEEDERS".GENERAL.MANUAL_SELECTED;
   #oLIMIT_RIGHT_LINE_2 := #_w2 AND #DATA.START_GENERAL_CONDITIONS AND #DATA.START_INITIAL_CONDITIONS_LINE_2 AND NOT #DATA.FEEDBACK_ON_LINE_2;
   #oLIMIT_LEFT_LINE_2 := #_w2 AND #DATA.STOP_GENERAL_CONDITIONS AND #DATA.STOP_INITIAL_CONDITIONS_LINE_2 AND NOT #DATA.FEEDBACK_OFF_LINE_2;
END_REGION

REGION Network 39: HMI ACTIONS / HMI Action
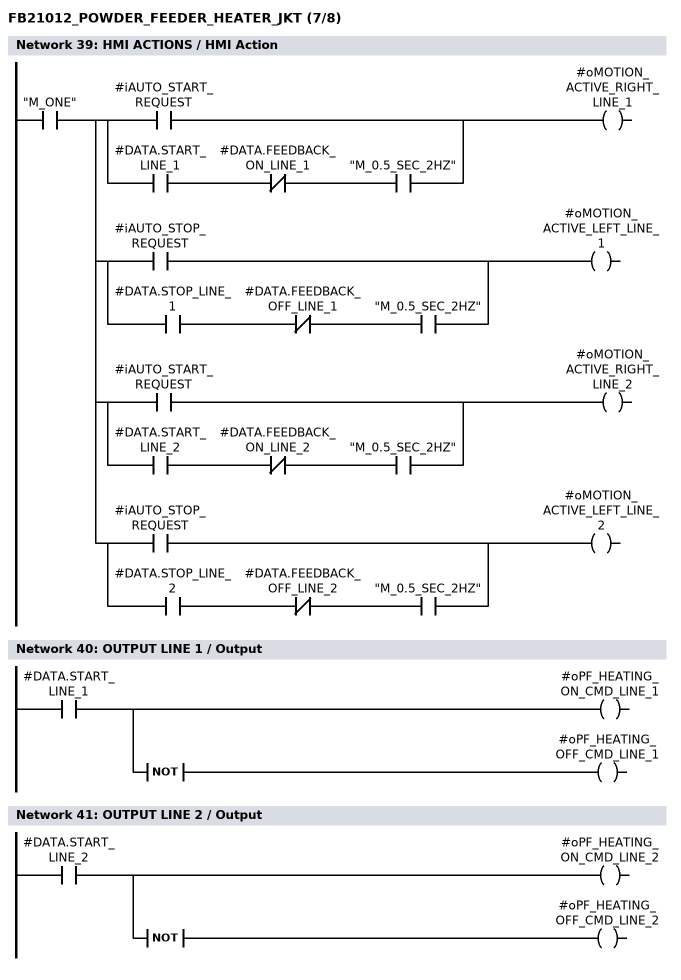
   RUNG wire#powerrail
      Contact( "M_ONE" )
      wire#w1
      Contact( #iAUTO_START_REQUEST )
      wire#w2
      Coil( #oMOTION_ACTIVE_RIGHT_LINE_1 )
   END_RUNG
   RUNG wire#w1
      Contact( #DATA.START_LINE_1 )
      I_Contact( #DATA.FEEDBACK_ON_LINE_1 )
      Contact( "M_0.5_SEC_2HZ" )
   END_RUNG wire#w2
   RUNG wire#w1
      Contact( #iAUTO_STOP_REQUEST )
      wire#w3
      Coil( #oMOTION_ACTIVE_LEFT_LINE_1 )
   END_RUNG
   RUNG wire#w1
      Contact( #DATA.STOP_LINE_1 )
      I_Contact( #DATA.FEEDBACK_OFF_LINE_1 )
      Contact( "M_0.5_SEC_2HZ" )
   END_RUNG wire#w3
   RUNG wire#w1
      Contact( #iAUTO_START_REQUEST )
      wire#w4
      Coil( #oMOTION_ACTIVE_RIGHT_LINE_2 )
   END_RUNG
   RUNG wire#w1
      Contact( #DATA.START_LINE_2 )
      I_Contact( #DATA.FEEDBACK_ON_LINE_2 )
      Contact( "M_0.5_SEC_2HZ" )
   END_RUNG wire#w4
   RUNG wire#w1
      Contact( #iAUTO_STOP_REQUEST )
      wire#w5
      Coil( #oMOTION_ACTIVE_LEFT_LINE_2 )
   END_RUNG
   RUNG wire#w1
      Contact( #DATA.STOP_LINE_2 )
      I_Contact( #DATA.FEEDBACK_OFF_LINE_2 )
      Contact( "M_0.5_SEC_2HZ" )
   END_RUNG wire#w5
   // the same network as SCL:
   #oMOTION_ACTIVE_RIGHT_LINE_1 := "M_ONE" AND (#iAUTO_START_REQUEST OR (#DATA.START_LINE_1 AND NOT #DATA.FEEDBACK_ON_LINE_1 AND "M_0.5_SEC_2HZ"));
   #oMOTION_ACTIVE_LEFT_LINE_1 := "M_ONE" AND (#iAUTO_STOP_REQUEST OR (#DATA.STOP_LINE_1 AND NOT #DATA.FEEDBACK_OFF_LINE_1 AND "M_0.5_SEC_2HZ"));
   #oMOTION_ACTIVE_RIGHT_LINE_2 := "M_ONE" AND (#iAUTO_START_REQUEST OR (#DATA.START_LINE_2 AND NOT #DATA.FEEDBACK_ON_LINE_2 AND "M_0.5_SEC_2HZ"));
   #oMOTION_ACTIVE_LEFT_LINE_2 := "M_ONE" AND (#iAUTO_STOP_REQUEST OR (#DATA.STOP_LINE_2 AND NOT #DATA.FEEDBACK_OFF_LINE_2 AND "M_0.5_SEC_2HZ"));
END_REGION

REGION Network 40: OUTPUT LINE 1 / Output
   RUNG wire#powerrail
      Contact( #DATA.START_LINE_1 )
      wire#w1
      Coil( #oPF_HEATING_ON_CMD_LINE_1 )
   END_RUNG
   RUNG wire#w1
      Not()
      Coil( #oPF_HEATING_OFF_CMD_LINE_1 )
   END_RUNG
   // the same network as SCL:
   #oPF_HEATING_ON_CMD_LINE_1 := #DATA.START_LINE_1;
   #oPF_HEATING_OFF_CMD_LINE_1 := NOT #DATA.START_LINE_1;
END_REGION

REGION Network 41: OUTPUT LINE 2 / Output
   RUNG wire#powerrail
      Contact( #DATA.START_LINE_2 )
      wire#w1
      Coil( #oPF_HEATING_ON_CMD_LINE_2 )
   END_RUNG
   RUNG wire#w1
      Not()
      Coil( #oPF_HEATING_OFF_CMD_LINE_2 )
   END_RUNG
   // the same network as SCL:
   #oPF_HEATING_ON_CMD_LINE_2 := #DATA.START_LINE_2;
   #oPF_HEATING_OFF_CMD_LINE_2 := NOT #DATA.START_LINE_2;
END_REGION

REGION Network 42: HEATER STATUS
   // STATUS:
   // 0: OFF WITH NO CONDITIONS
   // 1: ON
   // 2: OFF WITH CONDITIONS TO SWITCH ON
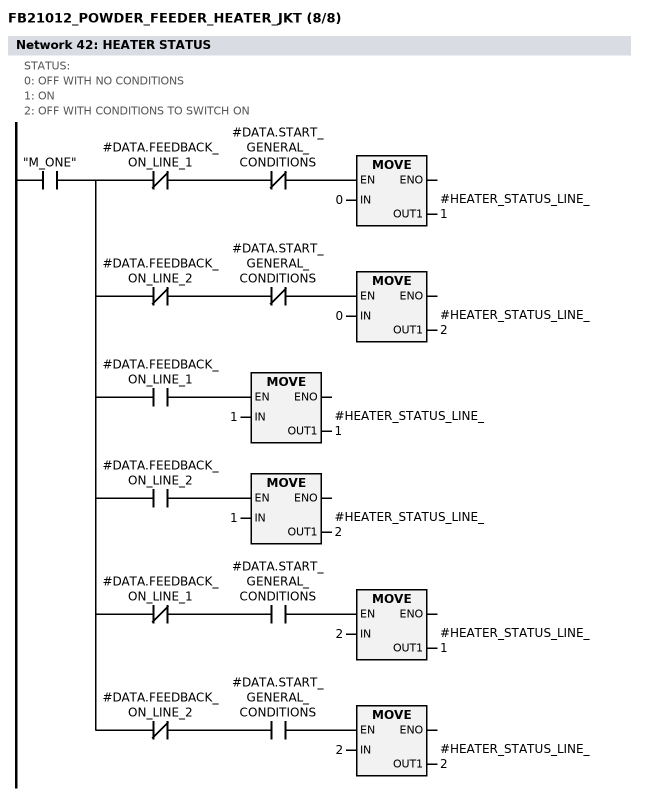
   RUNG wire#powerrail
      Contact( "M_ONE" )
      wire#w1
      I_Contact( #DATA.FEEDBACK_ON_LINE_1 )
      I_Contact( #DATA.START_GENERAL_CONDITIONS )
      Move(in := 0, out1 => #HEATER_STATUS_LINE_1)
   END_RUNG
   RUNG wire#w1
      I_Contact( #DATA.FEEDBACK_ON_LINE_2 )
      I_Contact( #DATA.START_GENERAL_CONDITIONS )
      Move(in := 0, out1 => #HEATER_STATUS_LINE_2)
   END_RUNG
   RUNG wire#w1
      Contact( #DATA.FEEDBACK_ON_LINE_1 )
      Move(in := 1, out1 => #HEATER_STATUS_LINE_1)
   END_RUNG
   RUNG wire#w1
      Contact( #DATA.FEEDBACK_ON_LINE_2 )
      Move(in := 1, out1 => #HEATER_STATUS_LINE_2)
   END_RUNG
   RUNG wire#w1
      I_Contact( #DATA.FEEDBACK_ON_LINE_1 )
      Contact( #DATA.START_GENERAL_CONDITIONS )
      Move(in := 2, out1 => #HEATER_STATUS_LINE_1)
   END_RUNG
   RUNG wire#w1
      I_Contact( #DATA.FEEDBACK_ON_LINE_2 )
      Contact( #DATA.START_GENERAL_CONDITIONS )
      Move(in := 2, out1 => #HEATER_STATUS_LINE_2)
   END_RUNG
   // the same network as SCL:
   IF "M_ONE" AND NOT #DATA.FEEDBACK_ON_LINE_1 AND NOT #DATA.START_GENERAL_CONDITIONS THEN
       #HEATER_STATUS_LINE_1 := 0;
   END_IF;
   IF "M_ONE" AND NOT #DATA.FEEDBACK_ON_LINE_2 AND NOT #DATA.START_GENERAL_CONDITIONS THEN
       #HEATER_STATUS_LINE_2 := 0;
   END_IF;
   IF "M_ONE" AND #DATA.FEEDBACK_ON_LINE_1 THEN #HEATER_STATUS_LINE_1 := 1; END_IF;
   IF "M_ONE" AND #DATA.FEEDBACK_ON_LINE_2 THEN #HEATER_STATUS_LINE_2 := 1; END_IF;
   IF "M_ONE" AND NOT #DATA.FEEDBACK_ON_LINE_1 AND #DATA.START_GENERAL_CONDITIONS THEN
       #HEATER_STATUS_LINE_1 := 2;
   END_IF;
   IF "M_ONE" AND NOT #DATA.FEEDBACK_ON_LINE_2 AND #DATA.START_GENERAL_CONDITIONS THEN
       #HEATER_STATUS_LINE_2 := 2;
   END_IF;
END_REGION
END_FUNCTION_BLOCK
